Fanuc KAREL source: compact_preamble.KL

PROGRAM KB00021
%NOLOCKGROUP
VAR
P1 : STRING[80];P2:INTEGER
BEGIN
P1='A'
P2=1
CLEAR(P1,P2)
END KB00021
